FUNCTION_BLOCK XtsCAGroup
VAR
END_VAR

METHOD AddMoverToGroup : BOOL
VAR_INPUT
END_VAR
END_METHOD

METHOD Enable : BOOL
VAR_INPUT
END_VAR
END_METHOD

END_FUNCTION_BLOCK

(* stored: Version 1.1.0.1, ProductVersion 3.1.4024.12
   POU XtsCAGroup: Id {7117239f-c04d-4613-b1bc-99efd400e059}, SpecialFunc None
   Method AddMoverToGroup: Id {ad749349-67a3-4a7b-bbde-0550486d46b8}
   Method Enable: Id {56f32a08-95f5-4aad-9a51-234b3e576357} *)
